FUNCTION_BLOCK JsonWriter IMPLEMENTS ITF_Writer
VAR
END_VAR

METHOD WriteMessage : BOOL
VAR_INPUT
	SomeString	: STRING(80);
END_VAR
ADSLOGSTR(msgCtrlMask := ADSLOG_MSGTYPE_LOG, msgFmtStr := 'I wrote a JSON line with: %s',strArg := SomeString);
END_METHOD

END_FUNCTION_BLOCK

(* stored: Version 1.1.0.1, ProductVersion 3.1.4024.12
   POU JsonWriter: Id {f665ae98-ed96-4d3d-9a09-fff139e1b7b7}, SpecialFunc None
   Method WriteMessage: Id {10cf58aa-9ece-4428-a808-5f378a1f06b3} *)
